TYPE VI : __System.VAR_INFO; END_TYPE

(* stored: Version 1.1.0.1, ProductVersion 3.1.4024.11
   DUT VI: Id {1d3aada1-a413-4388-b500-6efaa448d394} *)
